FUNCTION F_SetError : BOOL
VAR_INPUT
	nErrID	: INT;
	nLine	: INT;
END_VAR
VAR
END_VAR

IF nLine = 1 THEN
	bError1		:= TRUE;
ELSIF nLine = 2 THEN
	bError2		:= TRUE;
ELSIF nLine = 3 THEN
	bError1		:= TRUE;
	bError2		:= TRUE;
END_IF
nErrorID	:= nErrID;

END_FUNCTION

(* stored: Version 1.1.0.1, ProductVersion 3.1.4024.12
   POU F_SetError: Id {da17f6ed-e803-4727-8e3a-d1159d5d78ba}, SpecialFunc None *)
